// Slaapkamer 2 B1L0
TYPE ST_WP_Bedroom2 :
STRUCT
	fbButton1		: FB_DigitalIn;
END_STRUCT
END_TYPE

(* stored: Version 1.1.0.1, ProductVersion 3.1.4024.12
   DUT ST_WP_Bedroom2: Id {448db391-7f83-42b8-97fd-3fe5dec19610} *)
